{attribute 'linkalways'} 
{attribute 'no_explicit_call' := 'This FB is a CLASS and must be accessed using methods or properties'}
{attribute 'enable_dynamic_creation'}
FUNCTION_BLOCK Node_F_VN_VarianceFilter EXTENDS VisionNode
VAR
    ipSrcImage : _ITcVnImage;
    ipDestImage : _ITcVnImage;
    nKernelSize : _UDINT(0);
    hrPrev : _HRESULT(S_OK);
	hresult : _HRESULT(S_OK);
END_VAR

METHOD PUBLIC  Clone : I_Node
VAR
	pNode : POINTER TO Node_F_VN_VarianceFilter;
END_VAR
pNode := __NEW(Node_F_VN_VarianceFilter);
Clone := pNode^;
END_METHOD

METHOD FB_init : BOOL
VAR_INPUT
	bInitRetains : BOOL; // if TRUE, the retain variables are initialized (warm start / cold start)
	bInCopyCode : BOOL;  // if TRUE, the instance afterwards gets moved into the copy code (online change)
END_VAR
AddInput('ipSrcImage', ipSrcImage);
AddParameter('nKernelSize', nKernelSize);
AddInput('hrPrev', hrPrev);
AddOutput('ipDestImage', ipDestImage);
AddOutput('hresult',hresult);
END_METHOD

METHOD PROTECTED OnExecute
hresult.Value := F_VN_VarianceFilter(
    ipSrcImage := ipSrcImage.Value,
	ipDestImage := ipDestImage.Value,
    nKernelSize := nKernelSize.Value,
	hrPrev:= hrPrev.Value);
END_METHOD

METHOD PUBLIC PreExecutionCheck
VAR_INPUT
	Check : I_PreExecutionChecks;
END_VAR
Check.IsTrue(ipSrcImage.IsValid, 'ipSrcImage must contain an image');
Check.IsTrue(ipSrcImage.HasChannelCount(1), 'ipSrcImage must have 1 channel');
Check.IsTrue(ipSrcImage.IsPixelDepth(8), 'ipSrcImage must have 8 bit pixel depth');
END_METHOD

END_FUNCTION_BLOCK

(* stored: Version 1.1.0.1, ProductVersion 3.1.4024.13
   POU Node_F_VN_VarianceFilter: Id {5a819d45-bb00-0ca5-331a-aba7fffe8420}, SpecialFunc None
   Folder Constructor: Id {257f84ad-8648-083f-1260-5c9e5fe5a1f7}
   Method Clone: Id {9ea4789f-ef77-0e21-21f6-e3cf6415df5e}
   Method FB_init: Id {5d898af8-f9de-0ba7-117c-42e8ad88ea86}
   Method OnExecute: Id {67381b6a-76c6-019b-3f68-a83701b699f8}
   Method PreExecutionCheck: Id {898323b6-32b2-020d-1c6d-5c336187cdd8} *)
